INTERFACE IRecordDB

PROPERTY queue : REFERENCE TO dequeue
GET
END_GET
SET
END_SET
END_PROPERTY

END_INTERFACE

(* stored: Version 1.1.0.1, ProductVersion 3.1.4024.12
   Itf IRecordDB: Id {1d7da905-9dbc-4a62-9363-d7eaf62f12d7}
   Property queue: Id {18d54e9e-17bd-4a1e-8024-4a0247b3ade1}
   Get Get: Id {d1e55aac-b05f-4975-8355-8cb725db3b42}
   Set Set: Id {31f7b075-694c-4eea-b938-0dbf3bc2b8ab} *)
